{attribute addProperty BoxType "EL1808-0000-0016"}
{attribute addProperty Id "ChannelAT %I*ARRAY[0..7] OF Channel_E4AEF59E6480WcStateAT %I*WcState_98A4DF7520.250InfoDataAT %I*InfoData_192954DE1620"}
{attribute addProperty CRC "2007808796"}
{attribute addProperty SizeInBites "82"}
{attribute addProperty SizeInBytes "10.25"}
TYPE EL1808_772BB414 :
STRUCT
	{attribute addProperty Name "Channel"}
	Channel : ARRAY[0..7] OF Channel_E4AEF59E;
	{attribute addProperty Name "WcState"}
	WcState : WcState_98A4DF75;
	{attribute addProperty Name "InfoData"}
	InfoData : InfoData_192954DE;
END_STRUCT
END_TYPE

(* stored: Version 1.2.0.0, ProductVersion 3.1.4024.9
   DUT EL1808_772BB414: Id {13c2f896-7b68-4197-8727-72f895e5a207} *)
